KUKA KRL program: KRL_Prog.src, KRL_Prog.dat

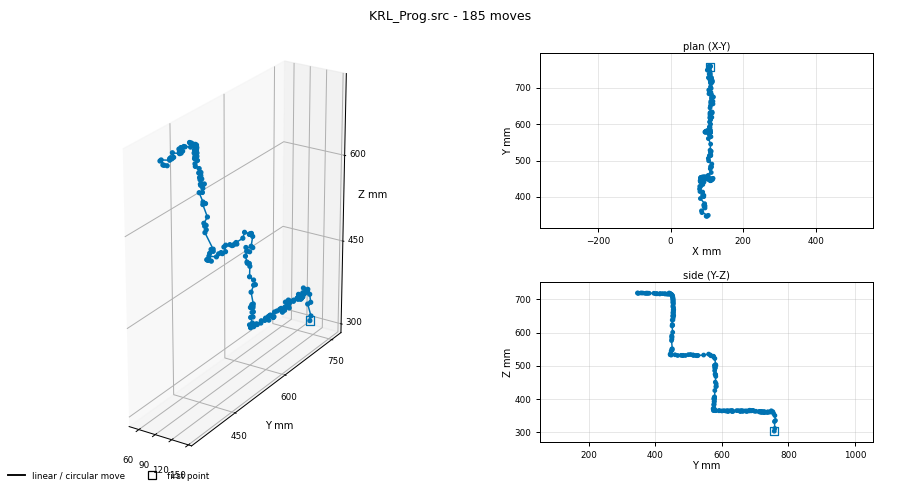
[picture p0: tool path of KRL_Prog.src, 185 of 185 moves have a stored position in this frame; points joined in program order, loops and branches not executed]
--- KRL_Prog.src ---
&ACCESS RVP
&REL 134
&PARAM TEMPLATE = C:\KRC\Roboter\Template\vorgabe
&PARAM EDITMASK = *
DEF baumerbalance( )
DECL RSIERR err
;FOLD INI
  ;FOLD BASISTECH INI
    GLOBAL INTERRUPT DECL 3 WHEN $STOPMESS==TRUE DO IR_STOPM ( )
    INTERRUPT ON 3
    BAS (#INITMOV,0 )
  ;ENDFOLD (BASISTECH INI)
  ;FOLD USER INI
    ;Make your modifications here

  ;ENDFOLD (USER INI)
;ENDFOLD (INI)

$APO.CVEL=4
$APO.CDIS=1
PTP {X 109.130, Y 757.730, Z 303.360, A -103.561, B -2.451, C 175.810}
LIN {X 110.150, Y 759.350, Z 311.640, A 11.603, B 4.834, C 179.568} C_DIS
LIN {X 104.230, Y 758.290, Z 332.420, A -142.222, B -4.530, C 178.258} C_DIS
LIN {X 108.222, Y 761.254, Z 335.407, A 40.980, B 4.426, C -178.008} C_DIS
LIN {X 107.060, Y 759.560, Z 350.470, A 53.256, B 3.902, C -177.113} C_DIS
LIN {X 104.700, Y 755.950, Z 356.100, A 122.816, B -1.349, C -175.338} C_DIS
LIN {X 106.870, Y 753.460, Z 361.840, A 38.874, B 4.496, C -178.171} C_DIS
LIN {X 101.187, Y 748.785, Z 364.710, A 175.419, B -4.523, C -178.239} C_DIS
LIN {X 106.402, Y 748.290, Z 361.804, A 119.747, B -1.097, C -175.272} C_DIS
LIN {X 108.557, Y 744.390, Z 360.943, A 93.379, B 1.122, C -175.278} C_DIS
LIN {X 108.790, Y 739.980, Z 360.700, A 39.190, B 4.486, C -178.147} C_DIS
LIN {X 106.313, Y 737.937, Z 361.539, A 172.069, B -4.413, C -177.978} C_DIS
LIN {X 109.077, Y 737.514, Z 360.252, A 78.182, B 2.322, C -175.738} C_DIS
LIN {X 108.590, Y 735.270, Z 360.120, A 58.489, B 3.623, C -176.769} C_DIS
LIN {X 104.168, Y 727.888, Z 362.246, A -176.035, B -4.734, C -178.930} C_DIS
LIN {X 111.970, Y 728.390, Z 359.550, A 35.523, B 4.595, C -178.437} C_DIS
LIN {X 108.658, Y 725.982, Z 361.182, A -164.354, B -4.852, C -179.909} C_DIS
LIN {X 112.370, Y 727.020, Z 359.860, A 54.014, B 3.864, C -177.061} C_DIS
LIN {X 108.470, Y 721.500, Z 362.030, A -163.762, B -4.853, C -179.960} C_DIS
LIN {X 113.067, Y 722.838, Z 360.418, A 44.376, B 4.301, C -177.749} C_DIS
LIN {X 109.603, Y 719.382, Z 362.002, A -166.244, B -4.847, C -179.750} C_DIS
LIN {X 114.190, Y 720.500, Z 360.490, A 38.700, B 4.502, C -178.185} C_DIS
LIN {X 109.672, Y 716.828, Z 362.244, A -162.533, B -4.853, C 179.937} C_DIS
LIN {X 114.600, Y 718.380, Z 360.620, A 39.043, B 4.491, C -178.158} C_DIS
LIN {X 110.036, Y 714.626, Z 362.356, A -161.844, B -4.852, C 179.878} C_DIS
LIN {X 114.980, Y 716.250, Z 360.700, A 39.958, B 4.461, C -178.087} C_DIS
$APO.CDIS = 0.983
LIN {X 110.512, Y 712.454, Z 362.366, A -176.451, B -4.726, C -178.896} C_DIS
LIN {X 112.280, Y 712.550, Z 361.510, A 75.797, B 2.498, C -175.838} C_DIS
$APO.CDIS = 1.000
LIN {X 109.910, Y 702.768, Z 363.356, A 114.306, B -0.643, C -175.190} C_DIS
LIN {X 111.742, Y 698.710, Z 363.302, A 35.723, B 4.590, C -178.421} C_DIS
LIN {X 105.140, Y 693.900, Z 365.790, A 168.249, B -4.269, C -177.689} C_DIS
LIN {X 107.215, Y 693.446, Z 365.079, A 86.568, B 1.675, C -175.445} C_DIS
LIN {X 106.860, Y 686.860, Z 365.770, A -167.408, B -4.841, C -179.651} C_DIS
LIN {X 110.932, Y 687.764, Z 364.514, A 38.038, B 4.522, C -178.237} C_DIS
LIN {X 105.690, Y 683.610, Z 366.400, A 165.064, B -4.134, C -177.455} C_DIS
LIN {X 112.600, Y 681.690, Z 364.210, A 93.879, B 1.081, C -175.269} C_DIS
LIN {X 112.994, Y 675.940, Z 364.364, A 167.339, B -4.231, C -177.621} C_DIS
LIN {X 118.000, Y 674.760, Z 362.690, A 38.384, B 4.512, C -178.210} C_DIS
LIN {X 112.626, Y 670.455, Z 364.442, A 75.803, B 2.498, C -175.838} C_DIS
LIN {X 110.554, Y 662.195, Z 365.048, A -173.349, B -4.779, C -179.153} C_DIS
LIN {X 116.573, Y 662.872, Z 362.865, A 40.490, B 4.443, C -178.046} C_DIS
LIN {X 110.670, Y 657.750, Z 365.310, A 162.644, B -4.023, C -177.283} C_DIS
LIN {X 116.720, Y 655.740, Z 362.460, A 37.505, B 4.538, C -178.279} C_DIS
LIN {X 109.795, Y 650.353, Z 365.057, A 78.105, B 2.328, C -175.741} C_DIS
LIN {X 108.625, Y 644.837, Z 365.183, A 90.762, B 1.337, C -175.334} C_DIS
LIN {X 108.780, Y 631.570, Z 365.230, A -161.079, B -4.849, C 179.814} C_DIS
LIN {X 114.340, Y 633.482, Z 362.934, A 36.076, B 4.580, C -178.393} C_DIS
LIN {X 108.660, Y 629.290, Z 365.050, A -164.633, B -4.852, C -179.886} C_DIS
LIN {X 114.617, Y 630.923, Z 362.533, A 42.718, B 4.364, C -177.874} C_DIS
LIN {X 108.623, Y 625.296, Z 364.989, A 84.017, B 1.877, C -175.524} C_DIS
LIN {X 107.857, Y 618.184, Z 364.971, A -172.490, B -4.791, C -179.224} C_DIS
LIN {X 113.572, Y 618.911, Z 362.549, A 38.699, B 4.502, C -178.185} C_DIS
LIN {X 109.170, Y 615.330, Z 364.340, A 107.923, B -0.102, C -175.148} C_DIS
LIN {X 110.210, Y 612.050, Z 364.100, A 63.338, B 3.337, C -176.475} C_DIS
LIN {X 107.308, Y 606.193, Z 365.044, A 115.101, B -0.709, C -175.199} C_DIS
LIN {X 110.092, Y 600.117, Z 364.286, A 65.869, B 3.178, C -176.331} C_DIS
LIN {X 106.718, Y 592.512, Z 365.216, A 152.050, B -3.456, C -176.590} C_DIS
LIN {X 108.631, Y 591.478, Z 364.808, A 74.942, B 2.560, C -175.876} C_DIS
LIN {X 106.043, Y 581.699, Z 365.837, A 176.946, B -4.568, C -178.360} C_DIS
LIN {X 108.160, Y 581.570, Z 365.100, A 54.641, B 3.832, C -177.019} C_DIS
LIN {X 105.070, Y 577.200, Z 365.630, A 121.421, B -1.235, C -175.306} C_DIS
LIN {X 106.537, Y 574.800, Z 365.570, A 28.878, B 4.745, C -178.979} C_DIS
LIN {X 105.140, Y 573.930, Z 370.600, A -149.473, B -4.713, C 178.843} C_DIS
LIN {X 109.070, Y 576.160, Z 373.970, A 13.649, B 4.846, C 179.741} C_DIS
LIN {X 106.180, Y 575.500, Z 383.230, A -152.791, B -4.772, C 179.117} C_DIS
LIN {X 109.570, Y 577.220, Z 384.240, A 16.341, B 4.853, C 179.968} C_DIS
LIN {X 108.020, Y 576.770, Z 392.110, A -155.889, B -4.813, C 179.376} C_DIS
LIN {X 109.874, Y 577.585, Z 393.213, A 19.076, B 4.849, C -179.800} C_DIS
LIN {X 105.420, Y 576.020, Z 400.250, A -153.435, B -4.782, C 179.171} C_DIS
LIN {X 108.948, Y 577.780, Z 400.170, A 23.601, B 4.818, C -179.419} C_DIS
LIN {X 106.670, Y 576.760, Z 402.620, A -150.820, B -4.739, C 178.954} C_DIS
LIN {X 108.982, Y 578.040, Z 402.932, A 23.485, B 4.819, C -179.429} C_DIS
LIN {X 107.360, Y 577.310, Z 405.410, A -149.205, B -4.708, C 178.821} C_DIS
LIN {X 109.202, Y 578.376, Z 406.561, A -1.430, B 4.613, C 178.490} C_DIS
LIN {X 104.742, Y 578.979, Z 425.643, A -122.795, B -3.695, C 176.851} C_DIS
LIN {X 107.540, Y 582.110, Z 437.330, A -148.565, B -4.695, C 178.768} C_DIS
LIN {X 109.850, Y 583.495, Z 438.196, A 9.366, B 4.813, C 179.380} C_DIS
LIN {X 106.770, Y 583.065, Z 445.654, A 23.220, B 4.822, C -179.451} C_DIS
LIN {X 100.897, Y 580.498, Z 450.831, A -30.509, B 3.300, C 176.440} C_DIS
LIN {X 100.530, Y 581.962, Z 468.196, A 26.736, B 4.779, C -179.157} C_DIS
LIN {X 97.030, Y 580.120, Z 473.340, A -151.070, B -4.744, C 178.974} C_DIS
LIN {X 99.734, Y 581.616, Z 473.012, A 26.066, B 4.789, C -179.212} C_DIS
LIN {X 96.432, Y 579.970, Z 475.340, A 31.591, B 4.691, C -178.756} C_DIS
LIN {X 94.510, Y 578.532, Z 485.590, A 168.755, B -4.289, C -177.727} C_DIS
LIN {X 96.824, Y 578.440, Z 494.517, A -149.503, B -4.714, C 178.845} C_DIS
LIN {X 100.780, Y 580.780, Z 493.700, A 30.242, B 4.719, C -178.866} C_DIS
LIN {X 95.854, Y 577.751, Z 501.050, A -154.748, B -4.800, C 179.281} C_DIS
LIN {X 105.595, Y 582.330, Z 501.273, A 25.247, B 4.800, C -179.281} C_DIS
LIN {X 103.280, Y 581.210, Z 503.550, A 135.257, B -2.323, C -175.738} C_DIS
LIN {X 107.373, Y 579.113, Z 522.061, A 51.649, B 3.982, C -177.223} C_DIS
LIN {X 104.720, Y 575.420, Z 526.742, A 169.411, B -4.315, C -177.776} C_DIS
LIN {X 107.580, Y 574.973, Z 528.757, A 96.105, B 0.896, C -175.230} C_DIS
LIN {X 108.510, Y 567.300, Z 530.180, A 143.520, B -2.912, C -176.116} C_DIS
LIN {X 111.125, Y 565.559, Z 532.297, A 35.179, B 4.604, C -178.465} C_DIS
LIN {X 104.050, Y 560.500, Z 535.200, A 113.337, B -0.561, C -175.179} C_DIS
LIN {X 110.320, Y 545.390, Z 532.330, A 85.049, B 1.796, C -175.491} C_DIS
LIN {X 108.714, Y 528.491, Z 531.066, A 137.583, B -2.494, C -175.836} C_DIS
LIN {X 111.850, Y 525.570, Z 530.310, A 50.657, B 4.029, C -177.293} C_DIS
LIN {X 109.660, Y 522.873, Z 530.900, A 98.225, B 0.718, C -175.200} C_DIS
LIN {X 110.620, Y 516.460, Z 531.370, A 36.219, B 4.576, C -178.382} C_DIS
LIN {X 106.748, Y 513.596, Z 532.562, A 179.449, B -4.635, C -178.561} C_DIS
LIN {X 110.630, Y 513.550, Z 531.900, A 47.838, B 4.157, C -177.494} C_DIS
LIN {X 103.928, Y 506.068, Z 533.881, A 98.424, B 0.702, C -175.198} C_DIS
LIN {X 104.850, Y 499.540, Z 533.430, A 134.467, B -2.264, C -175.706} C_DIS
LIN {X 113.480, Y 490.550, Z 531.090, A 64.651, B 3.256, C -176.399} C_DIS
LIN {X 110.060, Y 483.330, Z 531.550, A 165.854, B -4.168, C -177.513} C_DIS
LIN {X 112.772, Y 482.616, Z 530.664, A 55.955, B 3.762, C -176.932} C_DIS
LIN {X 109.350, Y 477.510, Z 531.500, A 104.142, B 0.218, C -175.152} C_DIS
LIN {X 111.898, Y 467.220, Z 531.029, A 43.076, B 4.351, C -177.847} C_DIS
LIN {X 103.482, Y 459.286, Z 533.178, A 111.008, B -0.364, C -175.161} C_DIS
LIN {X 108.840, Y 445.470, Z 533.660, A -159.960, B -4.845, C 179.719} C_DIS
LIN {X 115.184, Y 447.789, Z 532.126, A 30.784, B 4.708, C -178.822} C_DIS
$APO.CDIS = 1.000
LIN {X 111.017, Y 445.287, Z 533.351, A 25.469, B 4.797, C -179.262} C_DIS
LIN {X 109.520, Y 444.560, Z 534.460, A -146.266, B -4.642, C 178.581} C_DIS
$APO.CDIS = 1.000
LIN {X 111.765, Y 446.015, Z 535.717, A -84.584, B -0.953, C 175.241} C_DIS
LIN {X 112.325, Y 447.735, Z 544.343, A -143.793, B -4.576, C 178.382} C_DIS
LIN {X 116.710, Y 450.820, Z 547.490, A 18.887, B 4.850, C -179.816} C_DIS
LIN {X 113.602, Y 449.748, Z 550.334, A -153.399, B -4.781, C 179.168} C_DIS
LIN {X 116.410, Y 451.140, Z 550.950, A 11.023, B 4.829, C 179.519} C_DIS
LIN {X 103.406, Y 448.810, Z 575.909, A -140.980, B -4.492, C 178.160} C_DIS
LIN {X 105.030, Y 449.930, Z 580.510, A 12.297, B 4.839, C 179.626} C_DIS
LIN {X 102.641, Y 449.445, Z 586.054, A -149.188, B -4.708, C 178.819} C_DIS
LIN {X 104.520, Y 450.530, Z 587.360, A 19.088, B 4.849, C -179.799} C_DIS
LIN {X 101.244, Y 449.386, Z 590.450, A -143.027, B -4.554, C 178.322} C_DIS
LIN {X 105.726, Y 452.372, Z 600.649, A 16.535, B 4.853, C 179.985} C_DIS
LIN {X 99.000, Y 450.380, Z 620.070, A -151.273, B -4.747, C 178.991} C_DIS
LIN {X 102.580, Y 452.300, Z 621.840, A 18.159, B 4.852, C -179.878} C_DIS
LIN {X 98.898, Y 451.088, Z 623.910, A 3.481, B 4.725, C 178.890} C_DIS
LIN {X 92.277, Y 450.940, Z 637.610, A -153.402, B -4.781, C 179.168} C_DIS
LIN {X 96.621, Y 453.100, Z 638.140, A -68.876, B 0.374, C 175.161} C_DIS
LIN {X 96.923, Y 453.870, Z 644.750, A 15.817, B 4.852, C 179.924} C_DIS
LIN {X 93.762, Y 452.980, Z 649.020, A -157.655, B -4.830, C 179.525} C_DIS
LIN {X 96.145, Y 453.956, Z 649.204, A 20.707, B 4.841, C -179.663} C_DIS
LIN {X 93.268, Y 452.860, Z 650.800, A -155.568, B -4.809, C 179.349} C_DIS
LIN {X 98.696, Y 455.310, Z 651.580, A 17.642, B 4.852, C -179.922} C_DIS
LIN {X 92.445, Y 453.314, Z 657.760, A -154.508, B -4.797, C 179.260} C_DIS
LIN {X 94.810, Y 454.420, Z 659.060, A 18.445, B 4.851, C -179.854} C_DIS
LIN {X 91.641, Y 453.359, Z 661.018, A -135.932, B -4.313, C 177.772} C_DIS
LIN {X 93.102, Y 454.600, Z 664.070, A 13.802, B 4.847, C 179.754} C_DIS
LIN {X 89.885, Y 453.825, Z 667.897, A -151.662, B -4.754, C 179.023} C_DIS
LIN {X 92.790, Y 455.370, Z 668.770, A 11.710, B 4.835, C 179.577} C_DIS
LIN {X 90.031, Y 454.840, Z 674.580, A 19.494, B 4.847, C -179.765} C_DIS
LIN {X 84.553, Y 452.890, Z 677.550, A -16.676, B 4.055, C 177.331} C_DIS
LIN {X 83.695, Y 453.332, Z 681.419, A -160.878, B -4.849, C 179.796} C_DIS
LIN {X 87.326, Y 454.568, Z 687.096, A 22.044, B 4.832, C -179.550} C_DIS
LIN {X 83.245, Y 452.897, Z 689.712, A -172.078, B -4.796, C -179.259} C_DIS
LIN {X 83.776, Y 453.013, Z 692.978, A -158.221, B -4.834, C 179.572} C_DIS
LIN {X 86.690, Y 454.170, Z 693.710, A 23.868, B 4.815, C -179.397} C_DIS
LIN {X 82.902, Y 452.440, Z 698.771, A -156.726, B -4.821, C 179.446} C_DIS
LIN {X 86.895, Y 454.150, Z 699.110, A 27.847, B 4.762, C -179.064} C_DIS
LIN {X 83.707, Y 452.389, Z 703.598, A -165.984, B -4.848, C -179.772} C_DIS
LIN {X 86.776, Y 453.160, Z 704.550, A 52.246, B 3.953, C -177.182} C_DIS
LIN {X 85.954, Y 451.840, Z 707.880, A -164.640, B -4.852, C -179.885} C_DIS
LIN {X 87.871, Y 452.368, Z 708.416, A 33.117, B 4.656, C -178.631} C_DIS
LIN {X 84.760, Y 450.258, Z 711.569, A -164.594, B -4.852, C -179.889} C_DIS
LIN {X 87.849, Y 451.110, Z 711.730, A 23.631, B 4.818, C -179.416} C_DIS
LIN {X 83.445, Y 449.177, Z 712.647, A -172.474, B -4.791, C -179.226} C_DIS
LIN {X 88.932, Y 449.920, Z 713.490, A 30.161, B 4.721, C -178.873} C_DIS
LIN {X 84.526, Y 447.338, Z 714.856, A -174.067, B -4.768, C -179.093} C_DIS
LIN {X 88.284, Y 447.740, Z 715.260, A 24.909, B 4.804, C -179.309} C_DIS
$APO.CDIS = 0.991
LIN {X 81.355, Y 444.508, Z 716.990, A -169.828, B -4.822, C -179.448} C_DIS
LIN {X 83.299, Y 444.860, Z 717.150, A 66.143, B 3.161, C -176.316} C_DIS
$APO.CDIS = 1.000
LIN {X 82.024, Y 441.730, Z 718.890, A 175.383, B -4.522, C -178.236} C_DIS
LIN {X 91.927, Y 440.846, Z 715.366, A 28.729, B 4.747, C -178.991} C_DIS
LIN {X 87.628, Y 438.490, Z 715.750, A 104.752, B 0.167, C -175.150} C_DIS
LIN {X 88.743, Y 434.163, Z 715.481, A 31.897, B 4.684, C -178.731} C_DIS
LIN {X 80.325, Y 428.920, Z 716.450, A 174.050, B -4.480, C -178.132} C_DIS
LIN {X 82.673, Y 428.680, Z 716.421, A 67.281, B 3.087, C -176.254} C_DIS
LIN {X 79.822, Y 421.838, Z 717.006, A 99.093, B 0.645, C -175.190} C_DIS
LIN {X 80.936, Y 414.890, Z 717.110, A 169.051, B -4.300, C -177.749} C_DIS
LIN {X 88.435, Y 413.418, Z 716.001, A 88.310, B 1.536, C -175.396} C_DIS
LIN {X 88.230, Y 404.870, Z 716.820, A 172.562, B -4.430, C -178.016} C_DIS
LIN {X 91.702, Y 404.415, Z 716.508, A 84.371, B 1.849, C -175.512} C_DIS
LIN {X 91.361, Y 400.850, Z 716.760, A 28.935, B 4.744, C -178.974} C_DIS
LIN {X 82.167, Y 395.760, Z 717.990, A 129.132, B -1.854, C -175.514} C_DIS
LIN {X 93.870, Y 381.460, Z 718.064, A 54.240, B 3.852, C -177.046} C_DIS
LIN {X 91.235, Y 377.811, Z 718.255, A 145.466, B -3.042, C -176.217} C_DIS
LIN {X 94.872, Y 375.310, Z 718.040, A 41.110, B 4.422, C -177.998} C_DIS
LIN {X 92.400, Y 373.144, Z 718.491, A 124.504, B -1.486, C -175.379} C_DIS
LIN {X 94.775, Y 369.605, Z 717.789, A 38.475, B 4.509, C -178.203} C_DIS
LIN {X 85.131, Y 361.940, Z 718.760, A 104.189, B -0.041, C 175.004} C_DIS
LIN {X 86.363, Y 356.966, Z 719.042, A 156.317, B 0.813, C 171.551} C_DIS
LIN {X 103.794, Y 349.550, Z 717.896, A 20.322, B -4.632, C -170.168} C_DIS
LIN {X 97.995, Y 347.170, Z 718.650, A 169.539, B -1.110, C 169.198} C_DIS
LIN {X 100.420, Y 346.680, Z 718.820, A 169.539, B -1.110, C 169.198} C_DIS

END

--- KRL_Prog.dat ---
&ACCESS RVP
&REL 134
&PARAM TEMPLATE = C:\KRC\Roboter\Template\vorgabe
&PARAM EDITMASK = *
DEFDAT  BAUMERBALANCE
;FOLD EXTERNAL DECLARATIONS;%{PE}%MKUKATPBASIS,%CEXT,%VCOMMON,%P
;FOLD BASISTECH EXT;%{PE}%MKUKATPBASIS,%CEXT,%VEXT,%P
EXT  BAS (BAS_COMMAND  :IN,REAL  :IN )
DECL INT SUCCESS
;ENDFOLD (BASISTECH EXT)
;FOLD USER EXT;%{E}%MKUKATPUSER,%CEXT,%VEXT,%P
;Make here your modifications

;ENDFOLD (USER EXT)
;ENDFOLD (EXTERNAL DECLERATIONS)

ENDDAT
